{attribute 'qualified_only'}
{attribute 'strict'}
TYPE E_SunSpec_PV_Error :
(
	eNoError := 0,
	eModbusTCPError := 1,
	eSunSpecError := 2,
	eSunSpecTooBigValueReceived := 3
);
END_TYPE

(* stored: Version 1.1.0.1, ProductVersion 3.1.4024.11
   DUT E_SunSpec_PV_Error: Id {99a7fc84-326f-46b6-90ef-7925e6a828ca} *)
